PROGRAM POU_1
VAR
	x:BOOL;
	y:BOOL;
     rr:BOOL;
	 ss:bool;
	counter: CTU;
	coun:WORD;
END_VAR

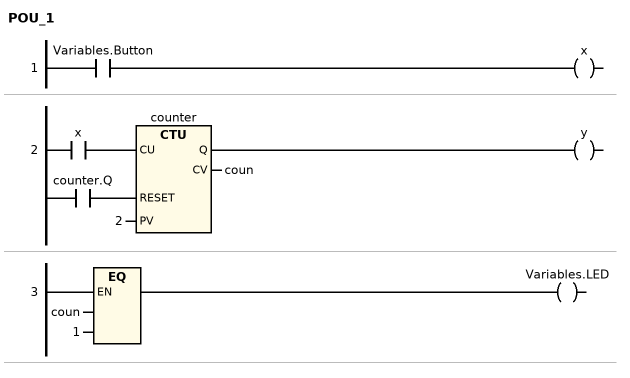
// NETWORK 1
x := Variables.Button;

// NETWORK 2
counter(CU := x, RESET := counter.Q, PV := 2, CV => coun); // CTU
y := counter.Q;

// NETWORK 3
Variables.LED := coun = 1;

END_PROGRAM

(* stored: Version 1.1.0.1, ProductVersion 3.1.4024.12
   POU POU_1: Id {4457e0b0-fcf5-4701-975e-7f7445db0e20}, SpecialFunc None *)
